(* IEC 61131-3 sources: eCockpitGit/test_project/src/%F%00 Library/%F%Common Functions/%F%UTF8, 3 files *)

(* ---- %POU%FU_CheckUTF8.st ---- *)
//This looks at an character and returns utf8 information about it
//It is not compatible with extended ascii (when all 8 bits are used)
// 0 means not utf-8 character
// 1 means start of utf-8 character
// 2 means middle of utf-8 character
// 3 means end of utf-8 character
// 4 means invalid
//It also returns the starting byte of the character
//To avoid cutting up utf 8 characters if this returns 1 or 2 when checking the end of a string, the string terminator should be moved to the start of the utf8 character
// |**Version**|**Author**| **Date** |**Changes**
// | 1         | NSN      | 06-12-20 | Creation
FUNCTION FU_CheckUTF8 : BYTE
VAR_INPUT
	strStart	:POINTER TO BYTE;		//Starting address of string to prevent underflow
	char		:POINTER TO BYTE;		//Character to check
END_VAR
VAR_OUTPUT
	start		:POINTER TO BYTE;		//Start of utf8 character
END_VAR
VAR
	i			:WORD;
END_VAR
(*%!%__DELIMITER__%!%*)
IF char <> 0 THEN
	IF char^.7 THEN
		IF char^.6 THEN
			FU_CheckUTF8		:=		1;
			start				:=		char;
		ELSE
			FOR i := 1 TO 6 DO
				char			:=		char - 1;
				IF char < strStart THEN
					RETURN;
				END_IF
				IF (char^ AND 2#11000000) = 192 THEN
					start		:=		char;
					IF char^.5 THEN
						IF char^.4 THEN
							IF char^.3 THEN
								IF char^.2 THEN
									IF char^.1 THEN
										FU_CheckUTF8			:=		4;
									ELSE
										IF i = 5 THEN
											FU_CheckUTF8		:=		3;
										ELSE
											FU_CheckUTF8		:=		2;
										END_IF
									END_IF
								ELSE
									IF i = 4 THEN
										FU_CheckUTF8		:=		3;
									ELSE
										FU_CheckUTF8		:=		2;
									END_IF
								END_IF
							ELSE
								IF i = 3 THEN
									FU_CheckUTF8		:=		3;
								ELSE
									FU_CheckUTF8		:=		2;
								END_IF
							END_IF
						ELSE
							IF i = 2 THEN
								FU_CheckUTF8		:=		3;
							ELSE
								FU_CheckUTF8		:=		2;
							END_IF
						END_IF
					ELSE
						IF i = 1 THEN
							FU_CheckUTF8		:=		3;
						ELSE
							FU_CheckUTF8		:=		2;
						END_IF
					END_IF
					RETURN;
				END_IF
			END_FOR
		END_IF
	ELSE
		FU_CheckUTF8			:=		0;
	END_IF
END_IF

(* ---- %POU%FU_FixUTF8.st ---- *)
//This fixes an utf8 string of fixed lenght
//Meaning it checks if the string cuts off in the middle of an utf8 string
// |**Version**|**Author**| **Date** |**Changes**
// | 1         | NSN      | 18-12-20 | Creation
FUNCTION FU_FixUTF8 : BOOL
VAR_INPUT
	str			:ANY;
END_VAR
VAR
	strPoint	:POINTER TO BYTE;
END_VAR
(*%!%__DELIMITER__%!%*)
CASE TO_BYTE(str.TypeClass) OF
	ESysType.tSTRING:
		strPoint			:=		str.pValue + TO_WORD(str.diSize) - 2;
ELSE
	strPoint				:=		str.pValue + TO_WORD(str.diSize) - 1;
END_CASE
IF strPoint^ <> 0 THEN
	CASE FU_CheckUTF8(strStart:=str.pValue,char:=strPoint, start=>str.pValue) OF
		1,2,4:str.pValue^	:=		0;
	END_CASE
END_IF

(* ---- %POU%FU_UTF8GetUnicode.st ---- *)
//This decodes an utf8 character and returns the unicode number
//Supports up to 6 byte encoding
//Returns 0 when invalid character is found
//Lenght of utf8 character is also returned, if the character is invalid, the length where ivalidity was found is returned.
// |**Version**|**Author**| **Date** |**Changes**
// | 1         | NSN      | 21-12-20 | Creation
FUNCTION FU_UTF8GetUnicode : DWORD
VAR_INPUT
	char		:POINTER TO BYTE;
END_VAR
VAR_OUTPUT
	len			:BYTE;
END_VAR
(*%!%__DELIMITER__%!%*)
IF char = 0 THEN
	FU_UTF8GetUnicode												:=		0;
END_IF
CASE char^ OF
	128..255:
		IF char^.6 THEN
			IF char^.5 THEN
				IF char^.4 THEN
					IF char^.3 THEN
						IF char^.2 THEN
							FU_UTF8GetUnicode						:=		SHL(TO_DWORD(char^ AND 2#00000011),30);
							char									:=		char + 1;
							IF char^.7 AND NOT char^.6 THEN
								FU_UTF8GetUnicode					:=		FU_UTF8GetUnicode OR SHL(TO_DWORD(char^ AND 2#00111111),24);
								char								:=		char + 1;
								IF char^.7 AND NOT char^.6 THEN
									FU_UTF8GetUnicode				:=		FU_UTF8GetUnicode OR SHL(TO_DWORD(char^ AND 2#00111111),18);
									char							:=		char + 1;
									IF char^.7 AND NOT char^.6 THEN
										FU_UTF8GetUnicode			:=		FU_UTF8GetUnicode OR SHL(TO_DWORD(char^ AND 2#00111111),12);
										char						:=		char + 1;
										IF char^.7 AND NOT char^.6 THEN
											FU_UTF8GetUnicode		:=		FU_UTF8GetUnicode OR SHL(TO_DWORD(char^ AND 2#00111111),6);
											char					:=		char + 1;
											IF char^.7 AND NOT char^.6 THEN
												FU_UTF8GetUnicode	:=		FU_UTF8GetUnicode OR (char^ AND 2#00111111);
												len					:=		6;
											ELSE	//Invalid utf returns 0
												FU_UTF8GetUnicode	:=		0;
												len					:=		5;
											END_IF
										ELSE	//Invalid utf returns 0
											FU_UTF8GetUnicode		:=		0;
											len						:=		4;
										END_IF
									ELSE	//Invalid utf returns 0
										FU_UTF8GetUnicode			:=		0;
										len							:=		3;
									END_IF
								ELSE	//Invalid utf returns 0
									FU_UTF8GetUnicode				:=		0;
									len								:=		2;
								END_IF
							ELSE	//Invalid utf returns 0
								FU_UTF8GetUnicode					:=		0;
								len									:=		1;
							END_IF
						ELSE	//5 byte encoding
							FU_UTF8GetUnicode						:=		SHL(TO_DWORD(char^ AND 2#00000011),24);
							char									:=		char + 1;
							IF char^.7 AND NOT char^.6 THEN
								FU_UTF8GetUnicode					:=		FU_UTF8GetUnicode OR SHL(TO_DWORD(char^ AND 2#00111111),18);
								char								:=		char + 1;
								IF char^.7 AND NOT char^.6 THEN
									FU_UTF8GetUnicode				:=		FU_UTF8GetUnicode OR SHL(TO_DWORD(char^ AND 2#00111111),12);
									char							:=		char + 1;
									IF char^.7 AND NOT char^.6 THEN
										FU_UTF8GetUnicode			:=		FU_UTF8GetUnicode OR SHL(TO_DWORD(char^ AND 2#00111111),6);
										char						:=		char + 1;
										IF char^.7 AND NOT char^.6 THEN
											FU_UTF8GetUnicode		:=		FU_UTF8GetUnicode OR (char^ AND 2#00111111);
												len					:=		5;
										ELSE	//Invalid utf returns 0
											FU_UTF8GetUnicode		:=		0;
											len						:=		4;
										END_IF
									ELSE	//Invalid utf returns 0
										FU_UTF8GetUnicode			:=		0;
										len							:=		3;
									END_IF
								ELSE	//Invalid utf returns 0
									FU_UTF8GetUnicode				:=		0;
									len								:=		2;
								END_IF
							ELSE	//Invalid utf returns 0
								FU_UTF8GetUnicode					:=		0;
								len									:=		1;
							END_IF
						END_IF
					ELSE	//4 byte encoding
						FU_UTF8GetUnicode							:=		SHL(TO_DWORD(char^ AND 2#00000111),18);
						char										:=		char + 1;
						IF char^.7 AND NOT char^.6 THEN
							FU_UTF8GetUnicode						:=		FU_UTF8GetUnicode OR SHL(TO_DWORD(char^ AND 2#00111111),12);
							char									:=		char + 1;
							IF char^.7 AND NOT char^.6 THEN
								FU_UTF8GetUnicode					:=		FU_UTF8GetUnicode OR SHL(TO_DWORD(char^ AND 2#00111111),6);
								char								:=		char + 1;
								IF char^.7 AND NOT char^.6 THEN
									FU_UTF8GetUnicode				:=		FU_UTF8GetUnicode OR (char^ AND 2#00111111);
									len								:=		4;
								ELSE	//Invalid utf returns 0
									FU_UTF8GetUnicode				:=		0;
									len								:=		3;
								END_IF
							ELSE	//Invalid utf returns 0
								FU_UTF8GetUnicode					:=		0;
								len									:=		2;
							END_IF
						ELSE	//Invalid utf returns 0
							FU_UTF8GetUnicode						:=		0;
							len										:=		1;
						END_IF
					END_IF
				ELSE	//3 byte encoding
					FU_UTF8GetUnicode								:=		SHL(TO_DWORD(char^ AND 2#00001111),12);
					char											:=		char + 1;
					IF char^.7 AND NOT char^.6 THEN
						FU_UTF8GetUnicode							:=		FU_UTF8GetUnicode OR SHL(TO_DWORD(char^ AND 2#00111111),6);
						char										:=		char + 1;
						IF char^.7 AND NOT char^.6 THEN
							FU_UTF8GetUnicode						:=		FU_UTF8GetUnicode OR (char^ AND 2#00111111);
							len										:=		3;
						ELSE	//Invalid utf returns 0
							FU_UTF8GetUnicode						:=		0;
							len										:=		2;
						END_IF
					ELSE	//Invalid utf returns 0
						FU_UTF8GetUnicode							:=		0;
						len											:=		1;
					END_IF
				END_IF
			ELSE	//2 byte encoding
				FU_UTF8GetUnicode									:=		SHL(TO_DWORD(char^ AND 2#00011111),6);
				char												:=		char + 1;
				IF char^.7 AND NOT char^.6 THEN
					FU_UTF8GetUnicode								:=		FU_UTF8GetUnicode OR (char^ AND 2#00111111);
					len												:=		2;
				ELSE	//Invalid utf returns 0
					FU_UTF8GetUnicode								:=		0;
					len												:=		1;
				END_IF
			END_IF
		ELSE	//Invalid utf returns 0
			FU_UTF8GetUnicode										:=		0;
			len														:=		1;
		END_IF
ELSE	//Characters in the ascii area
	FU_UTF8GetUnicode												:=		char^;
	len																:=		1;
END_CASE
